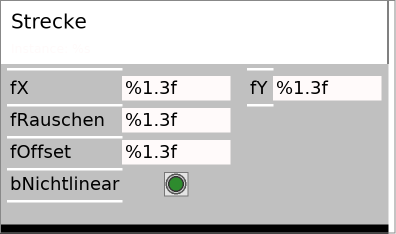
VISUALIZATION RET_VISU_Strecke  // 396x234
VAR_INPUT
   {attribute 'parameterstringof' := 'm_Input_FB'}
   m_Input_INST_Str : STRING;
END_VAR
VAR_IN_OUT
   m_Input_FB : Strecke;
END_VAR
    RoundedRectangle (0,0 388x81)
    RoundedRectangle (0,194 388x40)
    Rectangle (0,64 388x160)
    PushSwitch (164,172 24x24), variable: m_Input_FB.bNichtlinear, behaviour: TOGGLE, style: Switch-PushSwitch-Green
    Rectangle (8,8 388x27), "Strecke"
    Rectangle (8,35 388x27), "Instance: %s", text variable: m_Input_INST_Str
    Rectangle (7,68 115x2)
    Rectangle (122,76 108x24), "%1.3f", text variable: m_Input_FB.fX
        OnMouseClick: write the text variable via Default
    Rectangle (7,76 115x24), "fX"
    Rectangle (7,104 115x2)
    Rectangle (122,108 108x24), "%1.3f", text variable: m_Input_FB.fRauschen
        OnMouseClick: write the text variable via Default
    Rectangle (7,108 115x24), "fRauschen"
    Rectangle (7,136 115x2)
    Rectangle (122,140 108x24), "%1.3f", text variable: m_Input_FB.fOffset
        OnMouseClick: write the text variable via Default
    Rectangle (7,140 115x24), "fOffset"
    Rectangle (7,168 115x2)
    Rectangle (7,172 115x24), "bNichtlinear"
    Rectangle (7,200 115x2)
    Rectangle (247,68 26x2)
    Rectangle (273,76 108x24), "%1.3f", text variable: m_Input_FB.fY
    Rectangle (247,76 26x24), "fY"
    Rectangle (247,104 26x2)
END_VISUALIZATION

(* stored: Version 1.1.0.1, ProductVersion 3.1.4024.12
   Visu RET_VISU_Strecke: Id {ef5a617b-489c-4456-9dde-b841bd9f5e38} *)
